SUBAPPLICATION Uebung_074b_AUI (* RPTO auf UT ausgeben (Adapter Version) ohne Fendt-Schaltung *)
  (* Standard: 61499-2; Description: Copyright (c) 2023 Meisterschulen am Ostbahnhof This program and the accompanying materials are made available under the terms of the Eclipse Public License 2.0 which is available at https://www.eclipse.org/legal/epl-2.0/ SPDX-License-Identifier: EPL-2.0 *)
  (* Version 1.0, 2026-04-19, Franz Höpfinger, Meisterschulen am Ostbahnhof, initial API and implementation (Adapter Version of Uebung_074) *)
  PACKAGE Uebungen;
  IMPORT Uebungen::const::UT::TECU::DefaultPool_TECU::NumberVariable_Rear_PTO_output_shaft_speed;
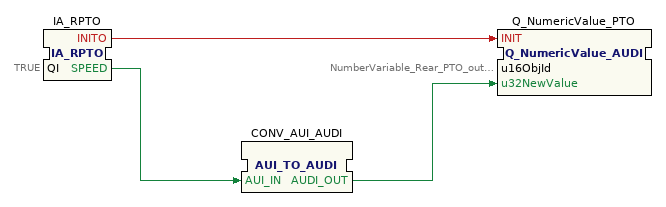
  FBS
    IA_RPTO : isobus::tecu::IA_RPTO(QI := TRUE);
    Q_NumericValue_PTO : isobus::UT::Q::Q_NumericValue_AUDI(u16ObjId := NumberVariable_Rear_PTO_output_shaft_speed);
    CONV_AUI_AUDI : adapter::conversion::unidirectional::AUI_TO_AUDI;
  END_FBS
  EVENT_CONNECTIONS
    IA_RPTO.INITO TO Q_NumericValue_PTO.INIT;
  END_CONNECTIONS
  ADAPTER_CONNECTIONS
    CONV_AUI_AUDI.AUDI_OUT TO Q_NumericValue_PTO.u32NewValue;
    IA_RPTO.SPEED TO CONV_AUI_AUDI.AUI_IN;
  END_CONNECTIONS
END_SUBAPPLICATION
